Staubli VAL3: find.pgx

public program find(string& x_sItem[], bool& x_bFound[])
begin
  //
  // find one item in the list
  //
  for i=0 to size(sSaveaxis)-1
    if sSaveaxis[i]==x_sItem
      x_bFound=true
      return
    endIf
  endFor
end
